FUNCTION_BLOCK VALFORMAT_21154F699884FA2C9 (* MBus device interface function block type *)
  (* Standard: 61499-2 *)
  (* Version 1.0, 09.09.2008, oberwal, nxtControl GmbH, Initial Version *)
  PACKAGE Main;
  (* Compiler Cpp *)
  {SET_ATTRIBUTE(Runtime.FBType.ImplementingType, Runtime.Standard#DYNGEN_VALFORMAT)}
  {SET_ATTRIBUTE(Configuration.GenericFBType.InterfaceParams, Runtime.Standard#I:=15;VALUE${I$}:INT,BYTE,INT,BYTE,INT,BYTE,STRING,BYTE,BOOL,BOOL,BOOL,BOOL,BOOL,BOOL,BOOL)}
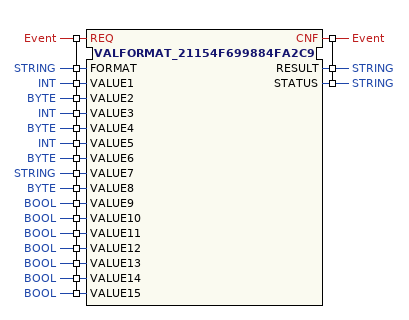
  EVENT_INPUT
    REQ WITH FORMAT, VALUE1, VALUE2, VALUE3, VALUE4, VALUE5, VALUE6, VALUE7, VALUE8, VALUE9, VALUE10, VALUE11, VALUE12, VALUE13, VALUE14, VALUE15; (* Request a formatting operation *)
  END_EVENT
  EVENT_OUTPUT
    CNF WITH RESULT, STATUS; (* Confirms a formattiong operation *)
  END_EVENT
  VAR_INPUT
    FORMAT : STRING; (* Defines a standard C printf like format *)
    VALUE1 : INT; (* A list of values to be converted into a string as defined in parameter FORMAT *)
    VALUE2 : BYTE; (* A list of values to be converted into a string as defined in parameter FORMAT *)
    VALUE3 : INT; (* A list of values to be converted into a string as defined in parameter FORMAT *)
    VALUE4 : BYTE; (* A list of values to be converted into a string as defined in parameter FORMAT *)
    VALUE5 : INT; (* A list of values to be converted into a string as defined in parameter FORMAT *)
    VALUE6 : BYTE; (* A list of values to be converted into a string as defined in parameter FORMAT *)
    VALUE7 : STRING; (* A list of values to be converted into a string as defined in parameter FORMAT *)
    VALUE8 : BYTE; (* A list of values to be converted into a string as defined in parameter FORMAT *)
    VALUE9 : BOOL; (* A list of values to be converted into a string as defined in parameter FORMAT *)
    VALUE10 : BOOL; (* A list of values to be converted into a string as defined in parameter FORMAT *)
    VALUE11 : BOOL; (* A list of values to be converted into a string as defined in parameter FORMAT *)
    VALUE12 : BOOL; (* A list of values to be converted into a string as defined in parameter FORMAT *)
    VALUE13 : BOOL; (* A list of values to be converted into a string as defined in parameter FORMAT *)
    VALUE14 : BOOL; (* A list of values to be converted into a string as defined in parameter FORMAT *)
    VALUE15 : BOOL; (* A list of values to be converted into a string as defined in parameter FORMAT *)
  END_VAR
  VAR_OUTPUT
    RESULT : STRING; (* The formatted result string *)
    STATUS : STRING; (* Error information *)
  END_VAR
  EC_STATES
    START;
  END_STATES
END_FUNCTION_BLOCK
